FUNCTION_BLOCK JsonNodeSettingsParser IMPLEMENTS I_NodeSettings
VAR
	parser : REFERENCE TO FB_JsonDomParser;
	baseJsonValue : SJsonValue;
	jsonLanguagePack : I_GraphDatatypes;
	
	propertyParser : JsonPropertySettingsParser(0);
	inputPortParser : JsonPortSettingsParser(0);
	outputPortParser : JsonPortSettingsParser(0);	
END_VAR

METHOD FB_init : BOOL
VAR_INPUT
	bInitRetains : BOOL; // if TRUE, the retain variables are initialized (warm start / cold start)
	bInCopyCode : BOOL;  // if TRUE, the instance afterwards gets moved into the copy code (online change)
	JsonLanguagePack : I_GraphDatatypes;
END_VAR
THIS^.jsonLanguagePack := JsonLanguagePack;

propertyParser.FB_init(bInitRetains, bInCopyCode, JsonLanguagePack);
inputPortParser.FB_init(bInitRetains, bInCopyCode, JsonLanguagePack);
outputPortParser.FB_init(bInitRetains, bInCopyCode, JsonLanguagePack);
END_METHOD

METHOD PUBLIC GetInputById : I_PortSettings
VAR_INPUT
	Id : PortId;
END_VAR
inputPortParser.Update(parser,GetInputObjectById(Id));
GetInputById := inputPortParser;
END_METHOD

METHOD PRIVATE GetInputObjectById : SJsonValue
VAR_INPUT
	Id : PortId;
END_VAR
GetInputObjectById := parser.GetArrayValueByIdx(GetInputsArray(),INT_TO_UDINT(Id));
END_METHOD

METHOD PRIVATE GetInputsArray : SJsonValue
GetInputsArray := parser.FindMember(baseJsonValue, 'inputs');
END_METHOD

METHOD PUBLIC GetOutputById : I_PortSettings
VAR_INPUT
	Id : PortId;
END_VAR
outputPortParser.Update(parser,GetOutputObjectById(Id));
GetOutputById := outputPortParser;
END_METHOD

METHOD PRIVATE GetOutputObjectById : SJsonValue
VAR_INPUT
	Id : PortId;
END_VAR
GetOutputObjectById := parser.GetArrayValueByIdx(GetOutputsArray(),INT_TO_UDINT(Id));
END_METHOD

METHOD PRIVATE GetOutputsArray : SJsonValue
GetOutputsArray := parser.FindMember(baseJsonValue, 'outputs');
END_METHOD

METHOD PRIVATE GetPropertiesObject : SJsonValue
GetPropertiesObject := parser.FindMember(baseJsonValue, 'properties');
END_METHOD

METHOD PUBLIC GetPropertyByIndex : I_ParameterSettings
VAR_INPUT
	Index : UDINT;
END_VAR
VAR
	i : UDINT;
	jsonIterator : SJsonIterator;
	jsonIteratorEnd : SJsonIterator;
END_VAR
jsonIterator := parser.MemberBegin(GetPropertiesObject());
jsonIteratorEnd := parser.MemberEnd(GetPropertiesObject());

FOR i := 0 TO Index DO
	IF i = Index THEN
		propertyParser.Update(parser,jsonIterator);
		GetPropertyByIndex := propertyParser;
		RETURN;
	END_IF
	
	IF jsonIterator = jsonIteratorEnd THEN
		RETURN;
	END_IF
	
	jsonIterator := parser.NextMember(jsonIterator);
END_FOR
END_METHOD

PROPERTY PUBLIC HasInputs : BOOL
GET
VAR
	jsonValue: SJsonValue;
END_VAR
jsonValue := GetInputsArray();

IF jsonValue = 0 THEN
	RETURN;	
END_IF

IF NOT parser.IsArray(jsonValue) THEN
	RETURN;
END_IF

HasInputs := TRUE;
END_GET
END_PROPERTY

PROPERTY PUBLIC HasOutputs : BOOL
GET
VAR
	jsonValue: SJsonValue;
END_VAR
jsonValue := GetOutputsArray();

IF jsonValue = 0 THEN
	RETURN;	
END_IF

IF NOT parser.IsArray(jsonValue) THEN
	RETURN;
END_IF

HasOutputs := TRUE;
END_GET
END_PROPERTY

PROPERTY PUBLIC HasProperties : BOOL
GET
HasProperties := PropertiesCount > 0;
END_GET
END_PROPERTY

PROPERTY PUBLIC Id : NodeId
GET
VAR
	jsonValue: SJsonValue;
END_VAR
jsonValue := parser.FindMember(baseJsonValue, 'id');
 
IF jsonValue = 0 THEN
	Id := -1;
	RETURN;	
END_IF

Id := DINT_TO_INT(parser.GetInt(jsonValue));
END_GET
END_PROPERTY

PROPERTY InputCount : UDINT
GET
IF NOT HasInputs THEN
	InputCount := 0;
END_IF

InputCount := parser.GetArraySize(GetInputsArray());
END_GET
END_PROPERTY

PROPERTY PUBLIC Mode : DINT
GET
VAR
	jsonValue: SJsonValue;
END_VAR
jsonValue := parser.FindMember(baseJsonValue, 'mode');
 
IF jsonValue = 0 THEN
	Mode := -1;
	RETURN;	
END_IF

Mode := parser.GetInt(jsonValue);
END_GET
END_PROPERTY

PROPERTY PUBLIC NodeType : T_MAXSTRING
GET
VAR
	jsonValue: SJsonValue;
END_VAR
jsonValue := parser.FindMember(baseJsonValue, 'type');
 
IF jsonValue = 0 THEN
	NodeType := '';
	RETURN;	
END_IF

NodeType := parser.GetString(jsonValue);
END_GET
END_PROPERTY

PROPERTY PUBLIC Order : DINT
GET
VAR
	jsonValue: SJsonValue;
END_VAR
jsonValue := parser.FindMember(baseJsonValue, 'order');
 
IF jsonValue = 0 THEN
	Order := -1;
	RETURN;	
END_IF

Order := parser.GetInt(jsonValue);
END_GET
END_PROPERTY

PROPERTY OutputCount : UDINT
GET
IF NOT HasOutputs THEN
	OutputCount := 0;
END_IF

OutputCount := parser.GetArraySize(GetOutputsArray());
END_GET
END_PROPERTY

PROPERTY PropertiesCount : UDINT
GET
VAR
	jsonIterator : SJsonIterator;
	jsonIteratorEnd : SJsonIterator;
END_VAR
jsonIterator := parser.MemberBegin(GetPropertiesObject());
jsonIteratorEnd := parser.MemberEnd(GetPropertiesObject());

WHILE jsonIterator <> jsonIteratorEnd DO
  jsonIterator := parser.NextMember(jsonIterator);
  PropertiesCount := PropertiesCount + 1;
END_WHILE
END_GET
END_PROPERTY

METHOD PUBLIC Update
VAR_INPUT
	Parser : REFERENCE TO FB_JsonDomParser;
	JsonValue : SJsonValue;
END_VAR
THIS^.parser REF= Parser;
THIS^.baseJsonValue := JsonValue;
END_METHOD

END_FUNCTION_BLOCK

(* stored: Version 1.1.0.1, ProductVersion 3.1.4024.12
   POU JsonNodeSettingsParser: Id {f1a26c4a-ea68-0e38-255b-514367792f9c}, SpecialFunc None
   Folder Constructor: Id {159144d5-e6c0-051b-3ad1-448b2d37afaf}
   Folder Private: Id {e758ed82-d627-0921-2203-e81f3e76808d}
   Method FB_init: Id {2678bb0f-405a-0143-3e9e-6f3a078a73bb}
   Method GetInputById: Id {8b509cf3-f068-0e02-351b-53a8bb60c15a}
   Method GetInputObjectById: Id {875bd275-8200-0d09-2ebe-abe489e7032f}
   Method GetInputsArray: Id {6023f5c1-40b7-0d48-0c94-f46658739782}
   Method GetOutputById: Id {01991eba-41f2-02eb-0621-3497916786ce}
   Method GetOutputObjectById: Id {50bc1f10-e42d-00f3-2bb7-fcf2c658a1e2}
   Method GetOutputsArray: Id {80e55ae0-8e59-06dd-16da-9c4772ced595}
   Method GetPropertiesObject: Id {0a150fcf-5b22-0b42-19c5-0fa8374b8d4e}
   Method GetPropertyByIndex: Id {9a6a3e5d-55de-0544-1c0b-03d386fffb0a}
   Property HasInputs: Id {c22b5ec9-8943-08b5-1b3a-845d2b516cad}
   Get Get: Id {bef5cbbf-9b95-0063-255b-071a27372ccb}
   Property HasOutputs: Id {ee4123ca-72d8-0129-2dd8-afcecca70580}
   Get Get: Id {34120d6f-a63f-0b74-1a30-b6ee93eae402}
   Property HasProperties: Id {cd858017-eaa7-0df2-031c-7cfa870c91aa}
   Get Get: Id {fe8dcb2b-a74a-06f0-15fc-54932f426768}
   Property Id: Id {55d0231f-d947-044a-1639-cbbbfccaa666}
   Get Get: Id {4b85e2e8-ecb4-0af1-216d-dc7ce532125e}
   Property InputCount: Id {85ba2751-5219-007a-3281-aebfeb7f9083}
   Get Get: Id {0204f34b-8cd0-0304-0f5e-fb1769e1714d}
   Property Mode: Id {85b5b2da-04f0-0824-0f7e-ca1c20c7427e}
   Get Get: Id {11dcbe7f-1466-0c5e-223d-75fd19ffbcb8}
   Property NodeType: Id {aaff5dba-64d5-02be-28a0-f681821ea0f5}
   Get Get: Id {d781155c-0602-05d7-25fe-b2414ea26a2b}
   Property Order: Id {7054a034-7329-010f-3b57-a6f9c20fba3b}
   Get Get: Id {5b0633f6-f42a-0618-2265-81edfec27aaa}
   Property OutputCount: Id {c7a1cc91-4450-0174-2774-d37c461c464e}
   Get Get: Id {9a9ed10a-c2c2-0137-09d7-0288975d23fb}
   Property PropertiesCount: Id {fcc32f86-e352-0ced-1481-206148ff0c57}
   Get Get: Id {c3d5f546-f516-0a0f-3944-05fb24465592}
   Method Update: Id {61bdb7ed-344f-083c-0280-18feabc53001} *)
